TYPE S_CONVEYORS :
STRUCT
	CONV0	: BIT;
	CONV1	: BIT;
	CONV2	: BIT;
	CONV3	: BIT;
	CONV4	: BIT;
	CONV5	: BIT;
	CONV6	: BIT;
	CONV7	: BIT;
END_STRUCT
END_TYPE

(* stored: Version 1.1.0.1, ProductVersion 3.1.4024.10
   DUT S_CONVEYORS: Id {5886a415-cfbb-4166-8d8c-73f8b14a00f3} *)
